// TIA Portal V20 export
FUNCTION "AccuS_Liter" : Void   // FC12, FBD
{ S7_Optimized_Access := 'TRUE' }
// stored: SetENOAutomatically false
   VAR_TEMP
      State : "Service_States";
   END_VAR
   VAR_TEMP   // added for the SCL form of the ladder/FBD networks
      _w1 : Bool;
   END_VAR
BEGIN

REGION Network 1
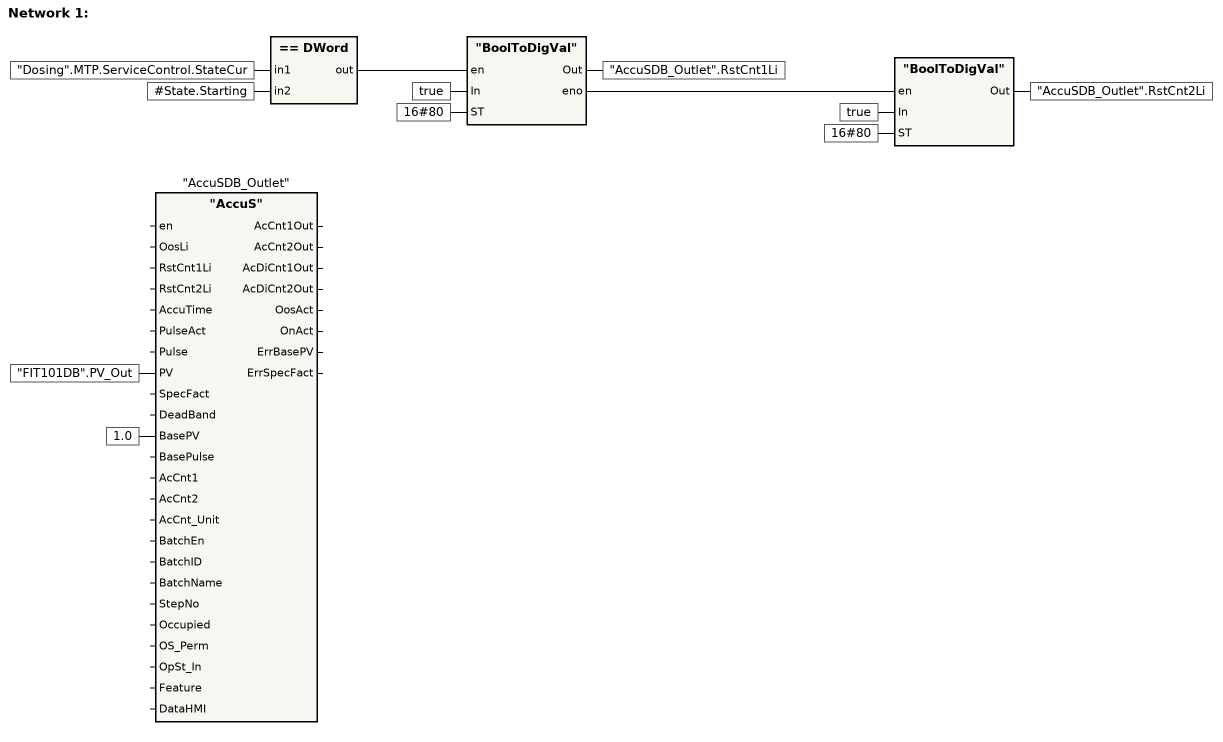
   "BoolToDigVal"(EN := "Dosing".MTP.ServiceControl.StateCur = #State.Starting,
                  In := true,
                  ST := 16#80,
                  Out => "AccuSDB_Outlet".RstCnt1Li,
                  ENO => #_w1);
   IF #_w1 THEN "BoolToDigVal"(In := true, ST := 16#80, Out => "AccuSDB_Outlet".RstCnt2Li); END_IF;
   "AccuSDB_Outlet"(PV := "FIT101DB".PV_Out, BasePV := 1.0);   // "AccuS"
END_REGION

REGION Network 2
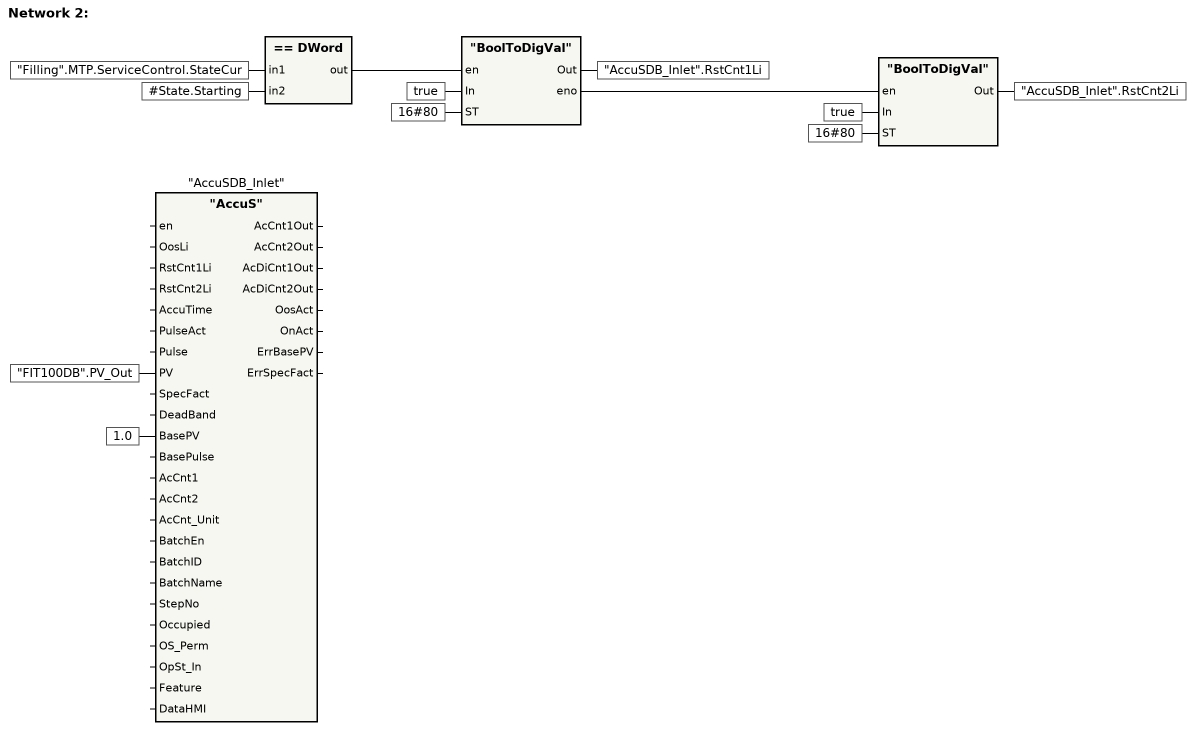
   "BoolToDigVal"(EN := "Filling".MTP.ServiceControl.StateCur = #State.Starting,
                  In := true,
                  ST := 16#80,
                  Out => "AccuSDB_Inlet".RstCnt1Li,
                  ENO => #_w1);
   IF #_w1 THEN "BoolToDigVal"(In := true, ST := 16#80, Out => "AccuSDB_Inlet".RstCnt2Li); END_IF;
   "AccuSDB_Inlet"(PV := "FIT100DB".PV_Out, BasePV := 1.0);   // "AccuS"
END_REGION
END_FUNCTION
